{attribute 'qualified_only'}
{attribute 'strict'}
{attribute 'to_string'}
TYPE E_ActionSelection :
(
	NONE := 0, //Nothing selected
	MOVE_TO_INFEED,
	MOVE_TO_CENTER,
	MOVE_TO_DOCKING,
	CENTER_TB
);
END_TYPE

(* stored: Version 1.1.0.1, ProductVersion 3.1.4024.12
   DUT E_ActionSelection: Id {6d5f3522-a992-4446-ba67-5780c65b3011} *)
